PROGRAM PRG_TEST
VAR
	fbTrafficLightTest : FB_TrafficLight_Test;
END_VAR

TcUnit.RUN();

END_PROGRAM

(* stored: Version 1.1.0.1, ProductVersion 3.1.4024.12
   POU PRG_TEST: Id {a0eda2ac-34e9-4306-912e-fa92d32909de}, SpecialFunc None *)
